TYPE ST_PNinput :
STRUCT
	PNIOBoxState		:	WORD;
	PNIOBoxDiag			:	WORD;	
	General 			: ST_PNInput_General;
	Battery				: ST_PNInput_Battery;
	Inputfield			: ST_PNInput_InputField;
	PSB					: ST_PNInput_PeakshaveBox;
	Powerstack			: ST_PNInput_Powerstack;
	GenControl 			: ST_PNInput_GenControl;
	InputGridControl	: ST_PNInput_InputGridControl;	
	ACDCCharger			: ST_PNInput_ACDCCharger;
END_STRUCT
END_TYPE

(* stored: Version 1.1.0.1, ProductVersion 3.1.4026.18
   DUT ST_PNinput: Id {5193972f-d452-482f-8515-bc8d6beb1a4f} *)
